{attribute addProperty BoxType "EK1122-0000-0018"}
{attribute addProperty Id "Beckhoff_AX2xxxsub_EK1100EK1100_179A0949162A_0001_AX2000_B110_0000AX2000_4A6B015820225.25"}
{attribute addProperty CRC "1605319744"}
{attribute addProperty SizeInBites "218"}
{attribute addProperty SizeInBytes "27.25"}
TYPE Beckhoff_AX2xxxEK1122_5FAF3C40 EXTENDS EK1122_179A0949 :
STRUCT
	{attribute addProperty Name "Beckhoff_AX2xxxsub_EK1100"}
	Beckhoff_AX2xxxsub_EK1100 : EK1100_179A0949;
	{attribute addProperty Name "A_0001_AX2000_B110_0000"}
	A_0001_AX2000_B110_0000 : AX2000_4A6B0158;
END_STRUCT
END_TYPE

(* stored: Version 1.2.0.0, ProductVersion 3.1.4024.9
   DUT Beckhoff_AX2xxxEK1122_5FAF3C40: Id {fe0f6336-2b47-4629-9f7e-226448a3f5f2} *)
